ABB RobotStudio station: saddlewelding_1dofpositioner.rspag

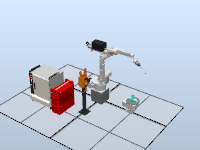
--- station ---
Station Final_1520_1dof (saved by RobotStudio 7.0.8743.626)
Controller 1520_simple_1dof_notmultimove, task T_ROB1: task frame (RAPID world) sits at (0, 0, 350) mm in the station
Controller 1520_simple_1dof_notmultimove
  mechanical unit ROB_1: IRB1520ID_4_150__02, 6 joints, base frame (0, 0, 0) mm
  mechanical unit M7DM1: MTD_250_M2009_REV1_01, 1 joints, base frame (1025, 0, 27) mm
Layout (positions relative to the parent item):
  - IRB1520ID_4_150__02 [mechanism, from Robots\IRB1520ID_4_150_G_02.rslib] at (0, 0, 350) mm; joint values [0, 0, 0, 0, 0.5236, 0] (rad or m)
  - Binzel_ID_22 [mechanism, from Tools\Binzel_ID_22.rslib] at (1056.21, 0, 1493) mm, rotated rx 180 ry 60 rz 180 deg
  - MTD_250_M2009_REV1_01 [mechanism] at (1025, 0, 377) mm; joint values [0] (rad or m)
      links: Base, Link1
  - saddle_simple_tpipe [part] at (1025, 0, 417) mm, rotated rx 90 ry 0 rz 0 deg
  - base [part]
  - IRC5_Singel-Cabinet [part, from Equipment\IRC5_Singel-Cabinet.rslib] at (-1110.18, -1000, 100) mm, rotated rx 90 ry 0 rz 0 deg
  - torch_cleaner_binzel [graphiccomponentgroup, from Equipment\Torch Cleaner Binzel.rslib] at (0, -692.97, 0) mm
    - Body 1 [part, from Equipment\Torch Cleaner Binzel.rslib]
    - Body 2 [part, from Equipment\Torch Cleaner Binzel.rslib]
    - Body 3 [part, from Equipment\Torch Cleaner Binzel.rslib]
    - Body 4 [part, from Equipment\Torch Cleaner Binzel.rslib]
    - Body 5 [part, from Equipment\Torch Cleaner Binzel.rslib]
    - Body 6 [part, from Equipment\Torch Cleaner Binzel.rslib]
    - Body 7 [part, from Equipment\Torch Cleaner Binzel.rslib]
    - Body 8 [part, from Equipment\Torch Cleaner Binzel.rslib]
    - Body 9 [part, from Equipment\Torch Cleaner Binzel.rslib]
    - Body 10 [part, from Equipment\Torch Cleaner Binzel.rslib]
    - Body 11 [part, from Equipment\Torch Cleaner Binzel.rslib]
    - Body 12 [part, from Equipment\Torch Cleaner Binzel.rslib]
  - Fronius_TPS4000_rev0 [part, from Equipment\Fronius_TPS4000.rslib] at (-561.29, -873.78, 0) mm, rotated rx 0 ry 0 rz 180 deg
  - Fronius_VR1500 [part, from Equipment\Fronius_VR1500.rslib] at (-229.13, 22.4, 164.6) mm
Attachment: Binzel_ID_22 is attached to IRB1520ID_4_150__02 / Link6
Attachment: saddle_simple_tpipe is attached to MTD_250_M2009_REV1_01 / Link1
Attachment: Fronius_VR1500 is attached to IRB1520ID_4_150__02 / Link3
Targets, tools, work objects and paths stored in the station and not in the controller backup, written as RAPID:
! task T_ROB1
MODULE Module1
  CONST robtarget Target_150_2:=[[5.512215763,-139.618372977,-304.487784237],[0.249807801,-0.286970556,-0.697531788,-0.607201257],[0,0,0,0],[9E+09,9E+09,9E+09,9E+09,9E+09,9E+09]];
  CONST robtarget Target_10_2:=[[3.533227121,139.843648253,-306.466772879],[0.257759887,0.281628821,-0.681799491,0.624014825],[0,0,0,0],[9E+09,9E+09,9E+09,9E+09,9E+09,9E+09]];
ENDMODULE


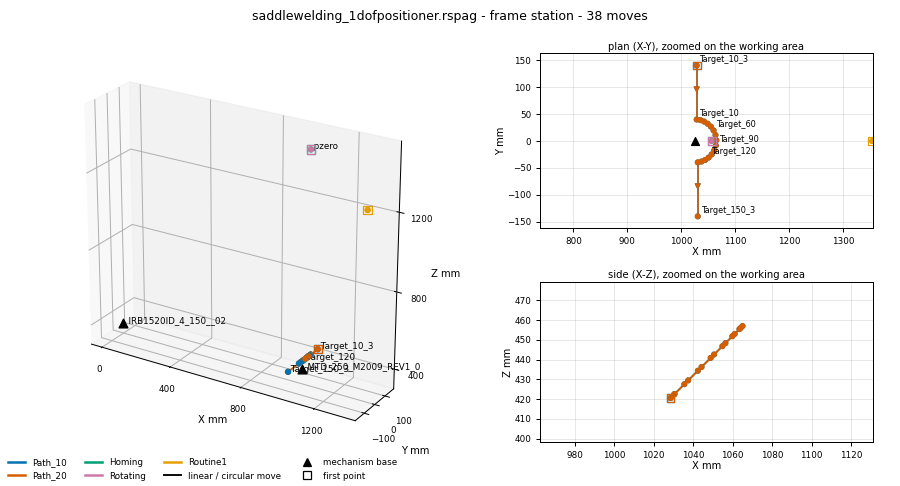
[picture p0: tool path of saddlewelding_1dofpositioner.rspag in frame station, 38 of 39 moves have a stored position in this frame; points joined in program order, loops and branches not executed]
--- Backups/1520_simple_1dof_notmultimove/RAPID/TASK1/PROGMOD/CalibData.mod ---
MODULE CalibData
	PERS tooldata tWeldGun:=[TRUE,[[49.841566361,0,372.194826196],[0.981627183,0,0.190808995,0]],[2,[0,0,100],[0,1,0,0],0,0,0]];
	TASK PERS wobjdata Workobject_1:=[FALSE,TRUE,"",[[1025,0,377],[1,0,0,0]],[[0,0,0],[1,0,0,0]]];
ENDMODULE

--- Backups/1520_simple_1dof_notmultimove/RAPID/TASK1/PROGMOD/Module1.mod ---
MODULE Module1
	CONST robtarget Target_10:=[[3.533227121,39.843648253,-306.466772879],[0.257759887,0.281628821,-0.681799491,0.624014825],[0,0,0,0],[0,9E+09,9E+09,9E+09,9E+09,9E+09]];
	CONST robtarget Target_20:=[[10.543230765,38.585493194,-299.456769235],[0.321420833,0.221566302,-0.701099521,0.596704687],[0,0,0,0],[0,9E+09,9E+09,9E+09,9E+09,9E+09]];
	CONST robtarget Target_30:=[[17.373721955,36.029901268,-292.626278045],[0.388755229,0.16472153,-0.714305049,0.55812587],[0,0,0,0],[0,9E+09,9E+09,9E+09,9E+09,9E+09]];
	CONST robtarget Target_40:=[[23.867766327,32.098749673,-286.132233673],[0.460189289,0.111711177,-0.721744598,0.50480805],[0,0,0,0],[0,9E+09,9E+09,9E+09,9E+09,9E+09]];
	CONST robtarget Target_50:=[[29.799997786,26.682581059,-280.200002214],[0.437744509,0.119413407,-0.78629609,0.419355029],[0,0,0,0],[0,9E+09,9E+09,9E+09,9E+09,9E+09]];
	CONST robtarget Target_60:=[[34.825013086,19.677867353,-275.174986914],[0.413718788,0.107673862,-0.848199495,0.312731068],[0,0,0,0],[0,9E+09,9E+09,9E+09,9E+09,9E+09]];
	CONST robtarget Target_70:=[[38.425796314,11.111173548,-271.574203686],[0.39293151,0.070355818,-0.899112857,0.179585518],[0,0,0,0],[0,9E+09,9E+09,9E+09,9E+09,9E+09]];
	CONST robtarget Target_80:=[[39.975373976,1.403380009,-270.024626024],[0.382849924,0.009483827,-0.923477587,0.022915929],[0,0,0,0],[0,9E+09,9E+09,9E+09,9E+09,9E+09]];
	CONST robtarget Target_90:=[[39.093432511,-8.467793958,-270.906567489],[0.388680804,-0.055130159,-0.909395508,-0.137432558],[0,0,0,0],[0,9E+09,9E+09,9E+09,9E+09,9E+09]];
	CONST robtarget Target_100:=[[36.006554193,-17.422056571,-273.993445807],[0.40726768,-0.099954989,-0.864160637,-0.278151811],[0,0,0,0],[0,9E+09,9E+09,9E+09,9E+09,9E+09]];
	CONST robtarget Target_110:=[[31.321421925,-24.87907813,-278.678578075],[0.431007099,-0.118376581,-0.804170506,-0.391828615],[0,0,0,0],[0,9E+09,9E+09,9E+09,9E+09,9E+09]];
	CONST robtarget Target_120:=[[25.602361861,-30.733028929,-284.397638139],[0.454215463,-0.11545924,-0.739906985,-0.482592096],[0,0,0,0],[0,9E+09,9E+09,9E+09,9E+09,9E+09]];
	CONST robtarget Target_130:=[[19.239246454,-35.069237173,-290.760753546],[0.381745973,-0.169334575,-0.731506947,-0.538974398],[0,0,0,0],[0,9E+09,9E+09,9E+09,9E+09,9E+09]];
	CONST robtarget Target_140:=[[12.485199881,-38.001576072,-297.514800119],[0.313796277,-0.226695714,-0.717409719,-0.579192752],[0,0,0,0],[0,9E+09,9E+09,9E+09,9E+09,9E+09]];
	CONST robtarget Target_150:=[[5.512215763,-39.618372977,-304.487784237],[0.249807801,-0.286970556,-0.697531788,-0.607201257],[0,0,0,0],[0,9E+09,9E+09,9E+09,9E+09,9E+09]];
	CONST robtarget pzero:=[[1056.205080757,0,1143],[0.5,0,0.866025404,0],[0,0,0,0],[0,9E+09,9E+09,9E+09,9E+09,9E+09]];

    CONST robtarget Target_10_r:=[[3.533227121,39.843648253,-306.466772879],[0.257759887,0.281628821,-0.681799491,0.624014825],[0,0,0,0],[180,9E+09,9E+09,9E+09,9E+09,9E+09]];
	CONST robtarget Target_20_r:=[[10.543230765,38.585493194,-299.456769235],[0.321420833,0.221566302,-0.701099521,0.596704687],[0,0,0,0],[180,9E+09,9E+09,9E+09,9E+09,9E+09]];
	CONST robtarget Target_30_r:=[[17.373721955,36.029901268,-292.626278045],[0.388755229,0.16472153,-0.714305049,0.55812587],[0,0,0,0],[180,9E+09,9E+09,9E+09,9E+09,9E+09]];
	CONST robtarget Target_40_r:=[[23.867766327,32.098749673,-286.132233673],[0.460189289,0.111711177,-0.721744598,0.50480805],[0,0,0,0],[180,9E+09,9E+09,9E+09,9E+09,9E+09]];
	CONST robtarget Target_50_r:=[[29.799997786,26.682581059,-280.200002214],[0.437744509,0.119413407,-0.78629609,0.419355029],[0,0,0,0],[180,9E+09,9E+09,9E+09,9E+09,9E+09]];
	CONST robtarget Target_60_r:=[[34.825013086,19.677867353,-275.174986914],[0.413718788,0.107673862,-0.848199495,0.312731068],[0,0,0,0],[180,9E+09,9E+09,9E+09,9E+09,9E+09]];
	CONST robtarget Target_70_r:=[[38.425796314,11.111173548,-271.574203686],[0.39293151,0.070355818,-0.899112857,0.179585518],[0,0,0,0],[180,9E+09,9E+09,9E+09,9E+09,9E+09]];
	CONST robtarget Target_80_r:=[[39.975373976,1.403380009,-270.024626024],[0.382849924,0.009483827,-0.923477587,0.022915929],[0,0,0,0],[180,9E+09,9E+09,9E+09,9E+09,9E+09]];
	CONST robtarget Target_90_r:=[[39.093432511,-8.467793958,-270.906567489],[0.388680804,-0.055130159,-0.909395508,-0.137432558],[0,0,0,0],[180,9E+09,9E+09,9E+09,9E+09,9E+09]];
	CONST robtarget Target_100_r:=[[36.006554193,-17.422056571,-273.993445807],[0.40726768,-0.099954989,-0.864160637,-0.278151811],[0,0,0,0],[180,9E+09,9E+09,9E+09,9E+09,9E+09]];
	CONST robtarget Target_110_r:=[[31.321421925,-24.87907813,-278.678578075],[0.431007099,-0.118376581,-0.804170506,-0.391828615],[0,0,0,0],[180,9E+09,9E+09,9E+09,9E+09,9E+09]];
	CONST robtarget Target_120_r:=[[25.602361861,-30.733028929,-284.397638139],[0.454215463,-0.11545924,-0.739906985,-0.482592096],[0,0,0,0],[180,9E+09,9E+09,9E+09,9E+09,9E+09]];
	CONST robtarget Target_130_r:=[[19.239246454,-35.069237173,-290.760753546],[0.381745973,-0.169334575,-0.731506947,-0.538974398],[0,0,0,0],[180,9E+09,9E+09,9E+09,9E+09,9E+09]];
	CONST robtarget Target_140_r:=[[12.485199881,-38.001576072,-297.514800119],[0.313796277,-0.226695714,-0.717409719,-0.579192752],[0,0,0,0],[180,9E+09,9E+09,9E+09,9E+09,9E+09]];
	CONST robtarget Target_150_r:=[[5.512215763,-39.618372977,-304.487784237],[0.249807801,-0.286970556,-0.697531788,-0.607201257],[0,0,0,0],[180,9E+09,9E+09,9E+09,9E+09,9E+09]];

    CONST robtarget pzero_rotated:=[[1056.205080757,0,1143],[0.5,0,0.866025404,0],[0,0,0,0],[180,9E+09,9E+09,9E+09,9E+09,9E+09]];
	CONST robtarget Target_10_3:=[[3.533227121,139.843648253,-306.466772879],[0.257759887,0.281628821,-0.681799491,0.624014825],[0,0,0,0],[0,9E+09,9E+09,9E+09,9E+09,9E+09]];
	CONST robtarget Target_150_3:=[[5.512215763,-139.618372977,-304.487784237],[0.249807801,-0.286970556,-0.697531788,-0.607201257],[0,0,0,0],[0,9E+09,9E+09,9E+09,9E+09,9E+09]];
	CONST robtarget Target_10_r_2:=[[3.533227121,139.843648253,-306.466772879],[0.257759887,0.281628821,-0.681799491,0.624014825],[0,0,0,0],[180,9E+09,9E+09,9E+09,9E+09,9E+09]];
	CONST robtarget Target_150_r_2:=[[5.512215763,-139.618372977,-304.487784237],[0.249807801,-0.286970556,-0.697531788,-0.607201257],[0,0,0,0],[180,9E+09,9E+09,9E+09,9E+09,9E+09]];


    !***********************************************************
    !
    ! Module:  Module1
    !
    ! Description:
    !   <Insert description here>
    !
    ! Author: firmi
    !
    ! Version: 1.0
    !
    !***********************************************************


    !***********************************************************
    !
    ! Procedure main
    !
    !   This is the entry point of your program
    !
    !***********************************************************
    PROC main()
        !Add your code here
        ActUnit M7DM1;
        Homing;
        Path_10;
        Homing;
        Rotating;
        Path_20;
        Rotating;
        DeactUnit M7DM1;
    ENDPROC
	PROC Path_10()
	    MoveL Target_10_3,v400,z0,tWeldGun\WObj:=Workobject_1;
	    MoveL Target_10,v50,z0,tWeldGun\WObj:=Workobject_1;
	    MoveL Target_20,v50,z0,tWeldGun\WObj:=Workobject_1;
	    MoveL Target_30,v50,z0,tWeldGun\WObj:=Workobject_1;
	    MoveL Target_40,v50,z0,tWeldGun\WObj:=Workobject_1;
	    MoveL Target_50,v50,z0,tWeldGun\WObj:=Workobject_1;
	    MoveL Target_60,v50,z0,tWeldGun\WObj:=Workobject_1;
	    MoveL Target_70,v50,z0,tWeldGun\WObj:=Workobject_1;
	    MoveL Target_80,v50,z0,tWeldGun\WObj:=Workobject_1;
	    MoveL Target_90,v50,z0,tWeldGun\WObj:=Workobject_1;
	    MoveL Target_100,v50,z0,tWeldGun\WObj:=Workobject_1;
	    MoveL Target_110,v50,z0,tWeldGun\WObj:=Workobject_1;
	    MoveL Target_120,v50,z0,tWeldGun\WObj:=Workobject_1;
	    MoveL Target_130,v50,z0,tWeldGun\WObj:=Workobject_1;
	    MoveL Target_140,v50,z0,tWeldGun\WObj:=Workobject_1;
	    MoveL Target_150,v50,z0,tWeldGun\WObj:=Workobject_1;
		MoveL Target_150_3,v50,z0,tWeldGun\WObj:=Workobject_1;
	ENDPROC
    PROC Path_20()
	    MoveL Target_10_r_2,v400,z0,tWeldGun\WObj:=Workobject_1;
	    MoveL Target_10_r,v50,z0,tWeldGun\WObj:=Workobject_1;
	    MoveL Target_20_r,v50,z0,tWeldGun\WObj:=Workobject_1;
	    MoveL Target_30_r,v50,z0,tWeldGun\WObj:=Workobject_1;
	    MoveL Target_40_r,v50,z0,tWeldGun\WObj:=Workobject_1;
	    MoveL Target_50_r,v50,z0,tWeldGun\WObj:=Workobject_1;
	    MoveL Target_60_r,v50,z0,tWeldGun\WObj:=Workobject_1;
	    MoveL Target_70_r,v50,z0,tWeldGun\WObj:=Workobject_1;
	    MoveL Target_80_r,v50,z0,tWeldGun\WObj:=Workobject_1;
	    MoveL Target_90_r,v50,z0,tWeldGun\WObj:=Workobject_1;
	    MoveL Target_100_r,v50,z0,tWeldGun\WObj:=Workobject_1;
	    MoveL Target_110_r,v50,z0,tWeldGun\WObj:=Workobject_1;
	    MoveL Target_120_r,v50,z0,tWeldGun\WObj:=Workobject_1;
	    MoveL Target_130_r,v50,z0,tWeldGun\WObj:=Workobject_1;
	    MoveL Target_140_r,v50,z0,tWeldGun\WObj:=Workobject_1;
	    MoveL Target_150_r,v50,z0,tWeldGun\WObj:=Workobject_1;
		MoveL Target_150_r_2,v50,z0,tWeldGun\WObj:=Workobject_1;
	ENDPROC
	PROC Homing()
	    MoveL pzero,v400,z0,tWeldGun\WObj:=wobj0;
	ENDPROC
    PROC Rotating()
	    MoveL pzero,v400,fine,tWeldGun\WObj:=wobj0;
	ENDPROC
	PROC Routine1()
		MoveAbsJ [[0,0,0,0,30,-2.28959E-7],[0,9E+9,9E+9,9E+9,9E+9,9E+9]]\NoEOffs, v200, z50, tWeldGun;
		MoveJ [[1353.61,-0.00,913.74],[0.325568,-1.50795E-9,0.945519,-1.31084E-9],[0,0,-1,0],[0,9E+9,9E+9,9E+9,9E+9,9E+9]], v200, z50, tWeldGun;
		MoveL [[1353.61,-0.00,913.74],[0.325568,-1.50795E-9,0.945519,-1.31084E-9],[0,0,-1,0],[0,9E+9,9E+9,9E+9,9E+9,9E+9]], v200, z50, tWeldGun;
	ENDPROC
ENDMODULE
